// TIA Portal V20 export
TYPE "typeCmHmiInterfaceSoftCamsideTapeFixStageAxisC"
// stored: Access Published, Namespace Unit1.Em4
   STRUCT
      pos00_tape1 : "LER_typeSoftCamPosition";
      pos01_tape2 : "LER_typeSoftCamPosition";
      pos02_tape3 : "LER_typeSoftCamPosition";
      pos03_tape4 : "LER_typeSoftCamPosition";
      pos04_posistion : "LER_typeSoftCamPosition";
      pos05_posistion : "LER_typeSoftCamPosition";
      pos06_posistion : "LER_typeSoftCamPosition";
      pos07_posistion : "LER_typeSoftCamPosition";
      pos08_posistion : "LER_typeSoftCamPosition";
      pos09_posistion : "LER_typeSoftCamPosition";
      pos10_posistion : "LER_typeSoftCamPosition";
      pos11_posistion : "LER_typeSoftCamPosition";
      pos12_posistion : "LER_typeSoftCamPosition";
      pos13_posistion : "LER_typeSoftCamPosition";
      pos14_posistion : "LER_typeSoftCamPosition";
      pos15_posistion : "LER_typeSoftCamPosition";
   END_STRUCT;
END_TYPE
